INTERFACE PUBLIC AbortingCommands

METHOD PUBLIC StateComplete
END_METHOD

END_INTERFACE

(* stored: Version 1.1.0.1, ProductVersion 3.1.4026.12
   Itf AbortingCommands: Id {d9a12bf1-10a0-0e97-0748-591bd5c252aa}
   Method StateComplete: Id {017d2983-b7e5-4445-82f6-ae0b5327024d} *)
